FUNCTION_BLOCK FB_CargarPieza_SFC

VAR_IN_OUT
	    TpoPinza: TIME;
END_VAR

VAR_INPUT
    // SFC-Flags
    SFCPause: BOOL;
    SFCReset: BOOL;
    
    // Indicadores de sincronizacion
    Ack: BOOL := TRUE;
    Execute: BOOL;
    
    // Entradas
    CargadorDetras : BOOL;
	CargadorDelante : BOOL;
	CargadorArriba : BOOL;
	CargadorAbajo : BOOL;  
END_VAR
VAR_OUTPUT
    // Indicadores de sincronizacion
    Done: BOOL;
    Ready: BOOL;
    
    // Salidas
    CargadorAvanza : BOOL;
	CargadorBaja : BOOL; 	
	CargadorCierra : BOOL;
END_VAR
VAR
END_VAR

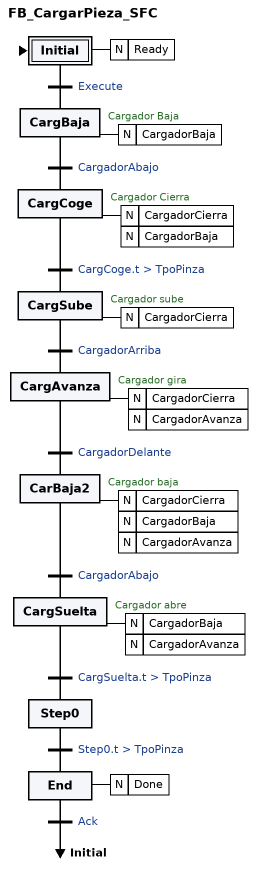
INITIAL_STEP Initial:
    Ready(N);
END_STEP
TRANSITION FROM Initial TO CargBaja
    := Execute;
END_TRANSITION
// Cargador Baja
STEP CargBaja:
    CargadorBaja(N);
END_STEP
TRANSITION FROM CargBaja TO CargCoge
    := CargadorAbajo;
END_TRANSITION
// Cargador Cierra
STEP CargCoge:
    CargadorCierra(N);
    CargadorBaja(N);
END_STEP
TRANSITION FROM CargCoge TO CargSube
    := CargCoge.t > TpoPinza;
END_TRANSITION
// Cargador sube
STEP CargSube:
    CargadorCierra(N);
END_STEP
TRANSITION FROM CargSube TO CargAvanza
    := CargadorArriba;
END_TRANSITION
// Cargador gira
STEP CargAvanza:
    CargadorCierra(N);
    CargadorAvanza(N);
END_STEP
TRANSITION FROM CargAvanza TO CarBaja2
    := CargadorDelante;
END_TRANSITION
// Cargador baja
STEP CarBaja2:
    CargadorCierra(N);
    CargadorBaja(N);
    CargadorAvanza(N);
END_STEP
TRANSITION FROM CarBaja2 TO CargSuelta
    := CargadorAbajo;
END_TRANSITION
// Cargador abre
STEP CargSuelta:
    CargadorBaja(N);
    CargadorAvanza(N);
END_STEP
TRANSITION FROM CargSuelta TO Step0
    := CargSuelta.t > TpoPinza;
END_TRANSITION
STEP Step0:
END_STEP
TRANSITION FROM Step0 TO End
    := Step0.t > TpoPinza;
END_TRANSITION
STEP End:
    Done(N);
END_STEP
TRANSITION FROM End TO Initial
    := Ack;
END_TRANSITION

END_FUNCTION_BLOCK

(* stored: Version 1.1.0.1, ProductVersion 3.1.4024.9
   POU FB_CargarPieza_SFC: Id {1f3006e8-5d97-40fb-a3f7-05d57d81639b}, SpecialFunc None *)
